(* CoDeSys 2.3 export: GLOBALE_VARIABLEN.EXP *)

(* Global variable list: Globale_Variablen *)
VAR_GLOBAL
	NetVarManager_Udp: NetVarManager_Udp_FB;

	g_bCPUStopNetVar : BOOL;
END_VAR
VAR_GLOBAL CONSTANT
	TELEGRAM_IDENT: DWORD := 16#33532D00;
END_VAR
